FUNCTION_BLOCK FB_EventLogger
VAR
	aEventBuffer : ARRAY[1..nBufferSize] OF ST_Event;
	nBufferIndex : INT := 0;
	_iCSVEventStorage : I_CSVEventStorage;	
END_VAR
VAR CONSTANT
	nBufferSize : INT := 255;
END_VAR

METHOD PUBLIC AddEvent : BOOL
VAR_IN_OUT
	stEvent : ST_Event;
END_VAR
IF NOT CheckEventBuffer() THEN
	nBufferIndex := nBufferIndex + 1;
	aEventBuffer[nBufferIndex].eEventType := stEvent.eEventType;
	aEventBuffer[nBufferIndex].eEventSeverity:= stEvent.eEventSeverity;
	aEventBuffer[nBufferIndex].nEventDefinition := stEvent.nEventDefinition;
	aEventBuffer[nBufferIndex].sEventMessage := stEvent.sEventMessage;
	F_EventTimeStamp(aEventBuffer[nBufferIndex]);
	AddEvent := TRUE;	
ELSE
	AddEvent := FALSE; 
END_IF

//Current event to be stored persistently
_iCSVEventStorage.StoreEvent(stEvent := aEventBuffer[nBufferIndex]);
END_METHOD

(*Returns True if event buffer full, False otherwise*)
METHOD PRIVATE CheckEventBuffer : BOOL
VAR_INPUT
END_VAR
IF (nBufferIndex + 1 > nBufferSize) THEN
	CheckEventBuffer := TRUE;
ELSE
	CheckEventBuffer := FALSE;
END_IF
END_METHOD

METHOD FB_init : BOOL
VAR_INPUT
	bInitRetains : BOOL; // if TRUE, the retain variables are initialized (warm start / cold start)
	bInCopyCode : BOOL;  // if TRUE, the instance afterwards gets moved into the copy code (online change)
	iCSVEventStorage : I_CSVEventStorage;
END_VAR
_iCSVEventStorage := iCSVEventStorage;
END_METHOD

END_FUNCTION_BLOCK

(* stored: Version 1.1.0.1, ProductVersion 3.1.4024.9
   POU FB_EventLogger: Id {4eea4031-622c-4f75-af55-a3cf5f6a3ee8}, SpecialFunc None
   Method AddEvent: Id {15e7c2bd-9dd2-496e-8af8-4b2cd3621b9e}
   Method CheckEventBuffer: Id {116f5a3d-bbf6-4d1d-b3a2-4918d4adfba1}
   Method FB_init: Id {55f63a4e-b746-4e36-89fe-444010d56774} *)
